// TIA Portal project "2022.05.16_指针化与创建模板" (V17)

(* hardware
DEVICE "S7-1500/ET200MP station_1"  S7-1500 station
   slot 0: "导轨_0"  Rack  6ES7 590-1***0-0AA0
   slot 1: "PLC_1500"  CPU 1516-3 PN/DP  6ES7 516-3AN00-0AB0  V1.7
      slot 3: "CPU 显示_1"  6ES7591-1BA00-0AA0
      slot 32768: "PROFINET 接口_1"  X1
         slot 32769: "端口_1"  X1 P1
         slot 32770: "端口_2"  X1 P2
      slot 33024: "PROFINET 接口_2"  X2
         slot 33025: "端口_1"  X2 P1
      slot 33280: "DP 接口_1"  X3
DEVICE "HMI_1"  TP1200 Comfort
   slot 0: "HMI_1"  TP1200 Comfort  6AV2 124-0MC01-0AX0  17.0.0.0
   slot 1: "HMI_RT_1"  TP1200 Comfort  6AV2 124-0MC01-0AX0  17.0.0.0
   slot 5: "HMI_1.IE_CP_1"  PROFINET Interface  17.0.0.0
      slot 1: "PROFINET Interface_1"  PROFINET Interface
         slot 1: "Port_1"  Port
         slot 2: "Port_2"  Port
   slot 7: "HMI_1.MPI/DP_CP_1"  MPI/DP Interface  17.0.0.0
*)

// ===== PLC "PLC_1500"  CPU 1516-3 PN/DP =====

DATA_BLOCK "数据块_1"   // DB1
{ S7_Optimized_Access := 'TRUE' }
VERSION : 0.1
   VAR
      索引变量 : Int;
      品牌 : Array[0..10] of String;
   END_VAR
BEGIN
END_DATA_BLOCK

ORGANIZATION_BLOCK "Main"   // OB1, LAD, ProgramCycle
TITLE = "Main Program Sweep (Cycle)"
{ S7_Optimized_Access := 'TRUE' }
VERSION : 0.1
   VAR_INPUT
      Initial_Call : Bool;   // Initial call of this OB
      Remanence : Bool;   // =True, if remanent data are available
   END_VAR
BEGIN
END_ORGANIZATION_BLOCK

(* ===== HMI "HMI_RT_1" =====
system functions are stored by id; their names below are inferred from use
connection "PLC_1500": ETHERNET, S7_1500_OMS
connection "Connection_1": ETHERNET, S7_1500_OMS

HMI tags "默认变量表"
   "Tag_ScreenNumber" : UInt, internal
   "指针化" : WString[254], internal
   "数据块_1_索引变量" : Int = PLC 数据块_1.索引变量, 1 s
   "数据块_1_品牌{0}" : String[254] = PLC 数据块_1.品牌[0], 1 s
   "数据块_1_品牌{1}" : String[254] = PLC 数据块_1.品牌[1], 1 s
   "数据块_1_品牌{2}" : String[254] = PLC 数据块_1.品牌[2], 1 s
   "数据块_1_品牌{3}" : String[254] = PLC 数据块_1.品牌[3], 1 s
   "数据块_1_品牌{4}" : String[254] = PLC 数据块_1.品牌[4], 1 s
   "数据块_1_品牌{5}" : String[254] = PLC 数据块_1.品牌[5], 1 s
   "数据块_1_品牌{6}" : String[254] = PLC 数据块_1.品牌[6], 1 s
   "数据块_1_品牌{7}" : String[254] = PLC 数据块_1.品牌[7], 1 s
   "数据块_1_品牌{8}" : String[254] = PLC 数据块_1.品牌[8], 1 s
   "数据块_1_品牌{9}" : String[254] = PLC 数据块_1.品牌[9], 1 s
   "数据块_1_品牌{10}" : String[254] = PLC 数据块_1.品牌[10], 1 s
   "指示灯控制1" : Bool AT %DB1.DBX0.0
   "指示灯控制2" : Bool AT %DB1.DBX0.0
   "指示灯控制3" : Bool AT %DB1.DBX0.0

screen "根画面" 1280x740, template "模板_1"
   on GenerateScreen: SetTag("Tag_ScreenNumber", 1)
   TextField "HmiScreenItemData" at 128,324 size 1024x27; Text '欢迎进入 HMI_1 (TP1200 Comfort)！'
   IOField "I/O 域_1" at 321,242 size 96x32; FormatPattern s99999
      ProcessValue <- "数据块_1_索引变量"
   IOField "I/O 域_2" at 326,303 size 96x32; FormatPattern ??????????
      ProcessValue <- "指针化"
   ScreenModuleView "按键指示灯_2" at 492,334 size 156x112; ScreenModuleType ""; Guid_{11997190-4463} '按钮松开'; Guid_{11997190-4465} '按钮按下'
      Guid_{11997190-4471} <- "指示灯控制1"
      on Guid_{11997190-4475}: InvertBit("指示灯控制1")
   ScreenModuleView "按键指示灯_1" at 308,432 size 156x112; ScreenModuleType ""; Guid_{11997190-4463} '按钮释放'; Guid_{11997190-4465} '按钮按下'; Guid_{11997190-4467} "FontList_C1440563122"
      Guid_{11997190-4471} <- "指示灯控制2"
      on Guid_{11997190-4475}: InvertBit("指示灯控制2")
   ScreenModuleView "按键指示灯_3" at 485,548 size 156x112; ScreenModuleType ""
      Guid_{11997190-4471} <- "指示灯控制3"
      on Guid_{11997190-4475}: InvertBit("指示灯控制3")

Template "模板_1" 1280x740
   Button "退出" at 1200,679 size 78x59; TextOff '退出'; PictureOff "ExitRuntime_TP1200_Comfort_TR"; PictureOn "ExitRuntime_TP1200_Comfort_TR"
      on Release: StopRuntime(0)
   Button "Template_Button" at 1120,679 size 78x59; TextOff 'Text'
   Button "Template_Button_1" at 1040,679 size 78x59; TextOff 'Text'
   Button "Template_Button_2" at 960,679 size 78x59; TextOff 'Text'
   Button "Template_Button_3" at 880,679 size 78x59; TextOff 'Text'
   Button "Template_Button_4" at 800,679 size 78x59; TextOff 'Text'
   Button "Template_Button_5" at 720,679 size 78x59; TextOff 'Text'
   Button "Template_Button_6" at 640,679 size 78x59; TextOff 'Text'
   Button "Template_Button_7" at 561,679 size 78x59; TextOff 'Text'
   Button "Template_Button_8" at 481,679 size 78x59; TextOff 'Text'
   Button "Template_Button_9" at 401,679 size 78x59; TextOff 'Text'
   Button "Template_Button_10" at 321,679 size 78x59; TextOff 'Text'
   Button "Template_Button_11" at 241,679 size 78x59; TextOff 'Text'
   Button "Template_Button_12" at 161,679 size 78x59; TextOff 'Text'
   Button "Template_Button_13" at 81,679 size 78x59; TextOff 'Text'
   Button "起始画面" at 1,679 size 78x59; TextOff '起始画面'; PictureOff "NavigateHome_TP1200_Comfort_TR"; PictureOn "NavigateHome_TP1200_Comfort_TR"
      on Release: ActivateScreen("根画面", 0)
*)

(* ===== HMI "HMI_RT_1" =====

ScreenModuleEditorView "按键指示灯" 640x480
   Button "按钮_1" at 10,66 size 156x56; TextOff 'Text'
*)

(* ===== HMI "HMI_RT_1" =====

ScreenModuleEditorView "按键指示灯" 640x480
   Button "按钮_1" at 10,66 size 156x56; TextOff 'Text'
      Appearance <- "Property_1"
*)

(* ===== HMI "HMI_RT_1" =====

ScreenModuleEditorView "按键指示灯" 640x480
   Button "按钮_1" at 10,66 size 156x56; TextOff 'Text'
      Appearance <- "Property_1"
*)